// TIA Portal V20 export
TYPE "UDT_BinAggr16"
TITLE = MTPDataObjectSUCLibrary/DataAssembly/ActiveElement/Aggr/Aggr16
   STRUCT
      WQC { ExternalWritable := 'False'} : Byte := 16#FF;   // Worst Quality Code variable
      OSLevel : Byte;   // OSLevel variable Operation Mode
      StateChannel { ExternalWritable := 'False'} : Bool;   // Selection of the active OperationMode interaction channel0: The operator switches (*Op) shall be used.1: The automatic switches (*Aut) shall be used.
      StateOffAut { ExternalWritable := 'False'} : Bool;   // Set OperationMode to Offline by automatic interaction (relevant, if StateChannel).1: OperationMode is set to Offline.0: no operation
      StateOpAut { ExternalWritable := 'False'} : Bool;   // Set OperationMode to Operator by automatic interaction (relevant, if StateChannel).1: OperationMode is set to Manual.0: no operation
      StateAutAut { ExternalWritable := 'False'} : Bool;   // Set OperationMode to Automatic by automatic interaction (relevant, if StateChannel).1: OperationMode is set to Automatic.0: no operation
      StateOffOp : Bool;   // Set OperationMode to Offline by operator interaction (relevant, if not StateChannel) 0-->1:request to set OperationMode to Offline 1-->0:acknowledge by PEA
      StateOpOp : Bool;   // Set OperationMode to Operator by operator interaction (relevant, if not StateChannel) 0-->1:request to set OperationMode to Manual 1-->0:acknowledge by PEA
      StateAutOp : Bool;   // Set OperationMode to Automatic by operator interaction (relevant, if not StateChannel) 0-->1:request to set OperationMode is to Automatic 1-->0:acknowledge by PEA
      StateOpAct { ExternalWritable := 'False'} : Bool;   // 1: current mode is Operator0: current mode is not Operator
      StateAutAct { ExternalWritable := 'False'} : Bool;   // 1: current mode is Automatic0: current mode is not Automatic
      StateOffAct { ExternalWritable := 'False'} : Bool;   // 1: current mode is Offline0: current mode is not Offline SourceMode for Number of CMs
      NoSrcChannel { ExternalWritable := 'False'} : Bool;   // Selection of the active OperationMode interaction channel number of CMs0: The operator switches (*Op) shall be used.1: The automatic switches (*Aut) shall be used.
      NoSrcIntAct { ExternalWritable := 'False'} : Bool;   // 1: current mode of units is Internal0: current mode of CMs is not Internal
      NoSrcIntAut { ExternalWritable := 'False'} : Bool;   // Set SourceMode to Internal by automatic interaction (relevant, if NoSrcChannel is true)1: SourceMode is set to Internal0: no operation
      NoSrcIntOp : Bool;   // Set SourceMode to Internal by operator interaction (relevant, if NoSrcChannel is false)0-->1:request to set OperationMode to Internal1-->0:acknowledge by PEA
      NoSrcManAct { ExternalWritable := 'False'} : Bool;   // 1: current mode is Manual0: current mode is not Manual
      NoSrcManAut { ExternalWritable := 'False'} : Bool;   // Set SourceMode to Manual by automatic interaction (relevant, if NoSrcChannel is true)1:SourceMode is set to Manual0:no operation
      NoSrcManOp : Bool;   // Set SourceMode to Manual by operator interaction (relevant, if NoSrcChannel is false)0-->1:request to set OperationMode to Manual1-->0 :acknowledge by PEA
      NoCMInt { ExternalWritable := 'False'} : Int;   // Internal Value (relevant, if NoSrcIntAct is false) Number CMs
      NoCMMan : Int;   // Manual Value (relevant, if NoSrcManAct is true) Number CMs SourceMode for Switch Mode
      SmSrcChannel { ExternalWritable := 'False'} : Bool;   // Selection of the active SourceMode interaction channel switch mode0:The operator switches (*Op) shall be used1:The automatic switches (*Aut) shall be used
      SmSrcIntAct { ExternalWritable := 'False'} : Bool;   // 1: current mode of units is Internal0: current mode of units is not Internal
      SmSrcIntAut { ExternalWritable := 'False'} : Bool;   // Set SourceMode to Internal by automatic interaction (relevant, if SrcChannelNo is true)1: SourceMode is set to Internal0: no operation
      SmSrcIntOp : Bool;   // Set SourceMode to Internal by operator interaction (relevant, if SmSrcChannel is false)0-->1:request to set OperationMode to Internal1-->0:acknowledge by PEA
      SmSrcManAct { ExternalWritable := 'False'} : Bool;   // 1: current mode is Manual0: current mode is not Manual
      SmSrcManAut { ExternalWritable := 'False'} : Bool;   // Set SourceMode to Manual by automatic interaction (relevant, if SmSrcChannel is true)1:SourceMode is set to Manual0:no operation
      SmSrcManOp : Bool;   // Set SourceMode to Manual by operator interaction (relevant, if SmSrcChannel is false)0-->1:request to set OperationMode to Manual1-->0 :acknowledge by PEA
      SmSrcManActTi { ExternalWritable := 'False'} : Bool;   // 1: current mode is Manual Time0: current mode is not Manual Time
      SmSrcManAutTi { ExternalWritable := 'False'} : Bool;   // Set SourceMode to Manual Time by automatic interaction (relevant, if SmSrcChannel is true)1:SourceMode is set to Manual Time0:no operation
      SmSrcManOpTi : Bool;   // Set SourceMode to Manual Time by operator interaction (relevant, if SmSrcChannel is false)0-->1:request to set OperationMode to Manual Time1-->0 :acknowledge by PEA
      MstrCMInt { ExternalWritable := 'False'} : Int;   // Internal Value (relevant, if SmSrcIntAct is true) Master CM
      MstrCMMan : Int;   // Manual Value (relevant, if SmSrcManAct is true) Master CM
      CMEn { ExternalWritable := 'False'} : DWord;   // Enables the CM 1-16 to be used by CM161: enabled0: disabled
      CMRdyToStart { ExternalWritable := 'False'} : DWord;   // Ready to use CM 1-16 Fbk1: CM is ready0: CM is not active
      CMFbkRun { ExternalWritable := 'False'} : DWord;   // Feedback signal CM 1-161: is running0: is not running
      CMCtrl { ExternalWritable := 'False'} : DWord;   // CM 1-16 Control by CM161: active (start)0: inactive (stop)
      OHCM01 { ExternalWritable := 'False'} : DWord;   // Operating hours CM 1
      OHCM02 { ExternalWritable := 'False'} : DWord;   // Operating hours CM 2
      OHCM03 { ExternalWritable := 'False'} : DWord;   // Operating hours CM 3
      OHCM04 { ExternalWritable := 'False'} : DWord;   // Operating hours CM 4
      OHCM05 { ExternalWritable := 'False'} : DWord;   // Operating hours CM 5
      OHCM06 { ExternalWritable := 'False'} : DWord;   // Operating hours CM 6
      OHCM07 { ExternalWritable := 'False'} : DWord;   // Operating hours CM 7
      OHCM08 { ExternalWritable := 'False'} : DWord;   // Operating hours CM 8
      OHCM09 { ExternalWritable := 'False'} : DWord;   // Operating hours CM 9
      OHCM10 { ExternalWritable := 'False'} : DWord;   // Operating hours CM 10
      OHCM11 { ExternalWritable := 'False'} : DWord;   // Operating hours CM 11
      OHCM12 { ExternalWritable := 'False'} : DWord;   // Operating hours CM 12
      OHCM13 { ExternalWritable := 'False'} : DWord;   // Operating hours CM 13
      OHCM14 { ExternalWritable := 'False'} : DWord;   // Operating hours CM 14
      OHCM15 { ExternalWritable := 'False'} : DWord;   // Operating hours CM 15
      OHCM16 { ExternalWritable := 'False'} : DWord;   // Operating hours CM 16
      PrioCM01 { ExternalWritable := 'False'} : Int;   // Switch On Priority for CM 1
      PrioCM02 { ExternalWritable := 'False'} : Int;   // Switch On Priority for CM 2
      PrioCM03 { ExternalWritable := 'False'} : Int;   // Switch On Priority for CM 3
      PrioCM04 { ExternalWritable := 'False'} : Int;   // Switch On Priority for CM 4
      PrioCM05 { ExternalWritable := 'False'} : Int;   // Switch On Priority for CM 5
      PrioCM06 { ExternalWritable := 'False'} : Int;   // Switch On Priority for CM 6
      PrioCM07 { ExternalWritable := 'False'} : Int;   // Switch On Priority for CM 7
      PrioCM08 { ExternalWritable := 'False'} : Int;   // Switch On Priority for CM 8
      PrioCM09 { ExternalWritable := 'False'} : Int;   // Switch On Priority for CM 9
      PrioCM10 { ExternalWritable := 'False'} : Int;   // Switch On Priority for CM 10
      PrioCM11 { ExternalWritable := 'False'} : Int;   // Switch On Priority for CM 11
      PrioCM12 { ExternalWritable := 'False'} : Int;   // Switch On Priority for CM 12
      PrioCM13 { ExternalWritable := 'False'} : Int;   // Switch On Priority for CM 13
      PrioCM14 { ExternalWritable := 'False'} : Int;   // Switch On Priority for CM 14
      PrioCM15 { ExternalWritable := 'False'} : Int;   // Switch On Priority for CM 15
      PrioCM16 { ExternalWritable := 'False'} : Int;   // Switch On Priority for CM 16
      OnAut { ExternalWritable := 'False'} : Bool;   // 1=On: On Command in Auto Mode
      OffAut { ExternalWritable := 'False'} : Bool;   // 1=Off: Off Command in Auto Mode
      OnOp : Bool;   // Set CM to On by Operator instruction (relevant, if StateOpAct)0-->1: request to set CM to On1-->0: acknowledge by PEA
      OffOp : Bool;   // Set CM to Off by Operator instruction (relevant, if StateOpAct)0-->1: request to set CM to Off1-->0: acknowledge by PEA
      OnAct { ExternalWritable := 'False'} : Bool;   // CM is set to On.1: CM is set to On.0: CM is not set to On.
      OffAct { ExternalWritable := 'False'} : Bool;   // CM is set to Off.1: CM is set to Off.0: CM is not set to Off.
      OpTimeSwMode { ExternalWritable := 'False'} : Bool;   // 0=Master aggregate / 1=Operating Time or Priority switch mode active
      PrefCMMode { ExternalWritable := 'False'} : Int;   // 1=Operating Time / 2=Priority switch mode active
      ChangeTime : Int;   // Time for Change the Master CM[h]
      MaxCM { ExternalWritable := 'False'} : Int;   // max. Number of CMs
      CMOn { ExternalWritable := 'False'} : DWord;   // CMs on Display
      CMAvail { ExternalWritable := 'False'} : DWord;   // CMs available Display
      NoCMRun { ExternalWritable := 'False'} : Int;   // Compared Number of CMs required/on
      ChangeTime_Out { ExternalWritable := 'False'} : DWord;   // Residual Time for Changing Master
   END_STRUCT;
END_TYPE
